FUNCTION_BLOCK FB_System_KKKW_Ablaufsteuerung
VAR_IN_OUT
	Zustand					: ST_System_KKKW_Zustand;
	Stellwert				: ST_System_KKKW_Stellwert;
	Steuerung				: ST_System_KKKW_Steuerung;
END_VAR
VAR_INPUT
	Zustand_Stellventil		: ST_SV_Zustand;
	Zustand_Pumpe			: ST_PU_Zustand;
END_VAR
VAR_OUTPUT
END_VAR
VAR
END_VAR

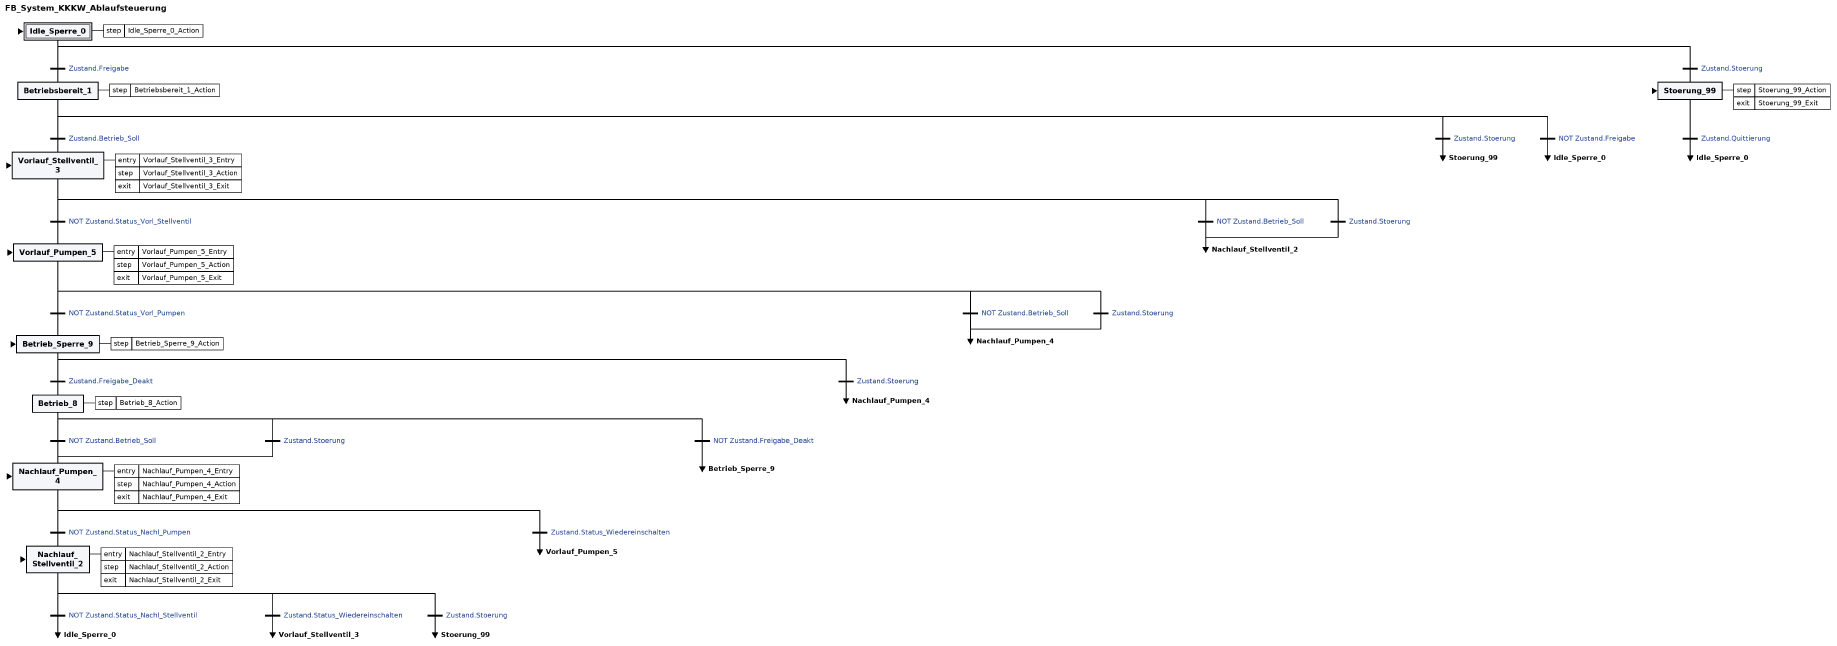
INITIAL_STEP Idle_Sperre_0:
    Idle_Sperre_0_Action(N);  // step action
END_STEP
TRANSITION FROM Idle_Sperre_0 TO Betriebsbereit_1
    := Zustand.Freigabe;
END_TRANSITION
TRANSITION FROM Idle_Sperre_0 TO Stoerung_99
    := Zustand.Stoerung;
END_TRANSITION
STEP Stoerung_99:
    Stoerung_99_Action(N);  // step action
    Stoerung_99_Exit(P0);  // exit action
END_STEP
TRANSITION FROM Stoerung_99 TO Idle_Sperre_0
    := Zustand.Quittierung;
END_TRANSITION
STEP Betriebsbereit_1:
    Betriebsbereit_1_Action(N);  // step action
END_STEP
TRANSITION FROM Betriebsbereit_1 TO Vorlauf_Stellventil_3
    := Zustand.Betrieb_Soll;
END_TRANSITION
TRANSITION FROM Betriebsbereit_1 TO Stoerung_99
    := Zustand.Stoerung;
END_TRANSITION
TRANSITION FROM Betriebsbereit_1 TO Idle_Sperre_0
    := NOT Zustand.Freigabe;
END_TRANSITION
STEP Vorlauf_Stellventil_3:
    Vorlauf_Stellventil_3_Entry(P1);  // entry action
    Vorlauf_Stellventil_3_Action(N);  // step action
    Vorlauf_Stellventil_3_Exit(P0);  // exit action
END_STEP
TRANSITION FROM Vorlauf_Stellventil_3 TO Vorlauf_Pumpen_5
    := NOT Zustand.Status_Vorl_Stellventil;
END_TRANSITION
TRANSITION FROM Vorlauf_Stellventil_3 TO Nachlauf_Stellventil_2
    := NOT Zustand.Betrieb_Soll;
END_TRANSITION
TRANSITION FROM Vorlauf_Stellventil_3 TO Nachlauf_Stellventil_2
    := Zustand.Stoerung;
END_TRANSITION
STEP Vorlauf_Pumpen_5:
    Vorlauf_Pumpen_5_Entry(P1);  // entry action
    Vorlauf_Pumpen_5_Action(N);  // step action
    Vorlauf_Pumpen_5_Exit(P0);  // exit action
END_STEP
TRANSITION FROM Vorlauf_Pumpen_5 TO Betrieb_Sperre_9
    := NOT Zustand.Status_Vorl_Pumpen;
END_TRANSITION
TRANSITION FROM Vorlauf_Pumpen_5 TO Nachlauf_Pumpen_4
    := NOT Zustand.Betrieb_Soll;
END_TRANSITION
TRANSITION FROM Vorlauf_Pumpen_5 TO Nachlauf_Pumpen_4
    := Zustand.Stoerung;
END_TRANSITION
STEP Betrieb_Sperre_9:
    Betrieb_Sperre_9_Action(N);  // step action
END_STEP
TRANSITION FROM Betrieb_Sperre_9 TO Betrieb_8
    := Zustand.Freigabe_Deakt;
END_TRANSITION
TRANSITION FROM Betrieb_Sperre_9 TO Nachlauf_Pumpen_4
    := Zustand.Stoerung;
END_TRANSITION
STEP Betrieb_8:
    Betrieb_8_Action(N);  // step action
END_STEP
TRANSITION FROM Betrieb_8 TO Nachlauf_Pumpen_4
    := NOT Zustand.Betrieb_Soll;
END_TRANSITION
TRANSITION FROM Betrieb_8 TO Nachlauf_Pumpen_4
    := Zustand.Stoerung;
END_TRANSITION
TRANSITION FROM Betrieb_8 TO Betrieb_Sperre_9
    := NOT Zustand.Freigabe_Deakt;
END_TRANSITION
STEP Nachlauf_Pumpen_4:
    Nachlauf_Pumpen_4_Entry(P1);  // entry action
    Nachlauf_Pumpen_4_Action(N);  // step action
    Nachlauf_Pumpen_4_Exit(P0);  // exit action
END_STEP
TRANSITION FROM Nachlauf_Pumpen_4 TO Nachlauf_Stellventil_2
    := NOT Zustand.Status_Nachl_Pumpen;
END_TRANSITION
TRANSITION FROM Nachlauf_Pumpen_4 TO Vorlauf_Pumpen_5
    := Zustand.Status_Wiedereinschalten;
END_TRANSITION
STEP Nachlauf_Stellventil_2:
    Nachlauf_Stellventil_2_Entry(P1);  // entry action
    Nachlauf_Stellventil_2_Action(N);  // step action
    Nachlauf_Stellventil_2_Exit(P0);  // exit action
END_STEP
TRANSITION FROM Nachlauf_Stellventil_2 TO Idle_Sperre_0
    := NOT Zustand.Status_Nachl_Stellventil;
END_TRANSITION
TRANSITION FROM Nachlauf_Stellventil_2 TO Vorlauf_Stellventil_3
    := Zustand.Status_Wiedereinschalten;
END_TRANSITION
TRANSITION FROM Nachlauf_Stellventil_2 TO Stoerung_99
    := Zustand.Stoerung;
END_TRANSITION

ACTION Betrieb_8_Action:
(* Stellwert setzen *)
Stellwert.Anford_Stellventil			:= TRUE;
Stellwert.Anford_Pumpe					:= TRUE;

(* Zustand setzen *)
Zustand.Status					:= E_System_KKKW_Zustand_Status_Betrieb;
END_ACTION

ACTION Betrieb_Sperre_9_Action:
(* Stellwert setzen *)
Stellwert.Anford_Stellventil		:= TRUE;
Stellwert.Anford_Pumpe				:= TRUE;


(* Zustand setzen *)
Zustand.Status				:= E_System_KKKW_Zustand_Status_Betrieb_Sperre;
END_ACTION

ACTION Betriebsbereit_1_Action:
(* Stellwert setzen *)
Stellwert.Anford_Stellventil	:= FALSE;
Stellwert.Anford_Pumpe			:= FALSE;

(* Zustand setzen *)
Zustand.Status			:= E_System_KKKW_Zustand_Status_Betriebsbereit;
END_ACTION

ACTION Idle_Sperre_0_Action:
(* Stellwert setzen *)
Stellwert.Anford_Stellventil		:= FALSE;
Stellwert.Anford_Pumpe		:= FALSE;

(* Zustand setzen *)
Zustand.Status				:= E_System_KKKW_Zustand_Status_Idle_Sperre;

(* Quittierungszustand auf False setzen, damit das System bei einer erneuten Störung nicht direkt wieder angeschaltet wird *)
Steuerung.Quittierung	:= FALSE;
END_ACTION

ACTION Nachlauf_Pumpen_4_Action:
(* Stellwert setzen *)
Stellwert.Anford_Stellventil			:= FALSE;
Stellwert.Anford_Pumpe					:= FALSE;

(* Zustand setzen *)
Zustand.Status						:= E_System_KKKW_Zustand_Status_Nachl_Pumpe;
Zustand.Status_Nachl_Pumpen			:= Zustand_Pumpe.Betrieb OR  Zustand_Pumpe.Status_Nachl;
Zustand.Status_Wiedereinschalten 	:= Zustand.Betrieb_Soll AND Stellwert.Einschalten;
END_ACTION

ACTION Nachlauf_Pumpen_4_Entry:
Zustand.Status_Nachl_Pumpen	:= TRUE;
END_ACTION

ACTION Nachlauf_Pumpen_4_Exit:
Zustand.Status_Nachl_Pumpen	:= FALSE;
END_ACTION

ACTION Nachlauf_Stellventil_2_Action:
(* Stellwert setzen *)
Stellwert.Anford_Stellventil		:= FALSE;
Stellwert.Anford_Pumpe				:= FALSE;

(* Zustand setzen *)
Zustand.Status						:= E_System_KKKW_Zustand_Status_Nachl_Stellventil;
Zustand.Status_Nachl_Stellventil	:= Zustand_Stellventil.Stellung OR Zustand_Stellventil.Stellungwechsel10;
Zustand.Status_Wiedereinschalten 	:= Zustand.Betrieb_Soll AND Stellwert.Einschalten;
END_ACTION

ACTION Nachlauf_Stellventil_2_Entry:
Zustand.Status_Nachl_Stellventil	:= TRUE;
END_ACTION

ACTION Nachlauf_Stellventil_2_Exit:
Zustand.Status_Nachl_Stellventil	:= FALSE;
END_ACTION

ACTION Stoerung_99_Action:
(* Stellwert setzen *)
Stellwert.Anford_Stellventil	:= FALSE;
Stellwert.Anford_Pumpe			:= FALSE;

(* Zustand setzen *)
Zustand.Stoerung				:= TRUE;
Zustand.Status					:= E_System_KKKW_Zustand_Status_Stoerung;
END_ACTION

ACTION Stoerung_99_Exit:
Zustand.Stoerung	:= FALSE;
END_ACTION

ACTION Vorlauf_Pumpen_5_Action:
(* Stellwert setzen *)
Stellwert.Anford_Stellventil		:= TRUE;
Stellwert.Anford_Pumpe		:= TRUE;

(* Zustand setzen *)
Zustand.Status				:= E_System_KKKW_Zustand_Status_Vorl_Pumpe;
Zustand.Status_Vorl_Pumpen	:= NOT(Zustand_Pumpe.Betrieb AND NOT Zustand_Pumpe.Status_Vorl);
END_ACTION

ACTION Vorlauf_Pumpen_5_Entry:
Zustand.Status_Vorl_Pumpen	:= TRUE;
END_ACTION

ACTION Vorlauf_Pumpen_5_Exit:
Zustand.Status_Vorl_Pumpen	:= FALSE;
END_ACTION

ACTION Vorlauf_Stellventil_3_Action:
(* Stellwert setzen *)
Stellwert.Anford_Stellventil		:= TRUE;
Stellwert.Anford_Pumpe				:= FALSE;

(* Zustand setzen *)
Zustand.Status				:= E_System_KKKW_Zustand_Status_Vorl_Stellventil;
Zustand.Status_Vorl_Stellventil	:= NOT(Zustand_Stellventil.Stellung AND NOT Zustand_Stellventil.Stellungwechsel01);
END_ACTION

ACTION Vorlauf_Stellventil_3_Entry:
Zustand.Status_Vorl_Stellventil	:= TRUE;
END_ACTION

ACTION Vorlauf_Stellventil_3_Exit:
Zustand.Status_Vorl_Stellventil	:= FALSE;
END_ACTION

END_FUNCTION_BLOCK

(* stored: Version 1.1.0.1, ProductVersion 3.1.4024.9
   POU FB_System_KKKW_Ablaufsteuerung: Id {f88aa24d-d292-41cd-97a6-0cb5dda30c17}, SpecialFunc None
   Action Betrieb_8_Action: Id {8b2e39c6-3501-425d-a516-194111b71cab}
   Action Betrieb_Sperre_9_Action: Id {8c033ef0-d9e2-4996-b7bb-b81efb957c8f}
   Action Betriebsbereit_1_Action: Id {1eeee31a-dd3f-4c81-95a0-e2afdd8b3db9}
   Action Idle_Sperre_0_Action: Id {8878baba-3ec4-4321-ab95-1344ab55e339}
   Action Nachlauf_Pumpen_4_Action: Id {388a68da-70bd-4819-b2ac-4ac4ffff015c}
   Action Nachlauf_Pumpen_4_Entry: Id {5abe7635-b517-461f-a6c2-9be970fffa66}
   Action Nachlauf_Pumpen_4_Exit: Id {4a553504-81bf-4237-9044-f604b53c890c}
   Action Nachlauf_Stellventil_2_Action: Id {7f7dc5f3-de4d-47d4-87fe-853732732db5}
   Action Nachlauf_Stellventil_2_Entry: Id {218a37ef-cdac-4f48-a598-e6bf68d914d1}
   Action Nachlauf_Stellventil_2_Exit: Id {d00be422-c533-4840-bc78-cc91fed88ec6}
   Action Stoerung_99_Action: Id {39c24e1b-ca0d-447f-9d1c-a5501fb7e213}
   Action Stoerung_99_Exit: Id {a165033e-1af9-4fc6-a55e-ff4f6e22db71}
   Action Vorlauf_Pumpen_5_Action: Id {67aabef7-49d5-41c4-ae02-dc1686cd95e0}
   Action Vorlauf_Pumpen_5_Entry: Id {3e573ff7-fd1e-42ae-9c86-6ac4bfa024a3}
   Action Vorlauf_Pumpen_5_Exit: Id {cde71ea0-25c7-4282-865e-295e6bc68251}
   Action Vorlauf_Stellventil_3_Action: Id {8c0d2185-620c-41c4-bdf4-a4ba4e23c65a}
   Action Vorlauf_Stellventil_3_Entry: Id {8c0232fd-59cd-4a07-98fd-3b03a86a8fbc}
   Action Vorlauf_Stellventil_3_Exit: Id {3aa63606-07e1-475a-b164-a4a0a8e7bd49} *)
